FUNCTION_BLOCK fbDatalogger
VAR_INPUT
	fData : LREAL;
END_VAR
VAR_OUTPUT
	afLog : ARRAY[0..999] OF LREAL;
	nLogJSTime : ULINT := 0;
END_VAR
VAR
	afCache : ARRAY[0..999] OF LREAL;
	nCount : DINT := 0;
	nPoints : DINT := 1000;
END_VAR

// Fill up the SampleArray
afCache[nCount] := fData;
// Increase the sampleIndex
nCount := nCount + 1;
IF nCount >= nPoints THEN
	// Copy values into log array
	afLog := afCache;
	// Increment log index to tell watching external logger the data has changed
	nLogJSTime := unixTime;
	// Reset count
	nCount := 0;
END_IF

END_FUNCTION_BLOCK

(* stored: Version 1.1.0.1, ProductVersion 3.1.0.36
   POU fbDatalogger: Id {7db4dd2a-609e-4033-9251-a25864602a12}, SpecialFunc None *)
